FUNCTION_BLOCK FB_ProductHandling
VAR CONSTANT
	sCycleStateTextDef: ARRAY[0..30]  OF STRING :=	
		['State 0: Wait for Start',
		'State 1: Gantry A, Gantry B and Product conveyor started',
		'State 2: ',
		'3',
		'4',
		'5',
		'6',
		'7',
		'8',
		'9',
		'State 10:',
		'State 11:',
		'State 12:',
		'State 13:',
		'State 14:',
		'State 15:',
		'State 16:',
		'State 17:',
		'State 18:',
		'State 19:',
		'State 20: Stopcylce waiting for EAMC ready',
		'State 21: Stop cycle awaiting gantries ready',
		'State 22: Stop cycle awaiting outfeed conveyor ready',
		'State 23: Stop cycle Stopping Gantries and conveyor',
		'State 24: Stop cycle awaiting restart',
		'State 25: Stop direct'];
	
	tCycleStateTimeouts: ARRAY[0..10] OF TIME := 
		[T#10S,T#10S,T#10S,T#10S,T#10S,T#10S,T#10S,T#10S,T#10S,T#10S,
		T#10S];

	sInitStateTextDef: ARRAY[0..10] OF STRING :=
		['State 0: Wait for Start',
		'State 1: Description Init State 1',
		'State 2: Description Init State 2',
		'State 3; Description Init State 3',
		'State 4; Description Init State 4',
		'State 5; Description Init State 5',
		'State 6; Error State'];

	tInitStateTimeouts: ARRAY[0..10] OF TIME := 
		[T#10S,T#10S,T#10S,T#10S,T#10S,T#10S,T#10S,T#10S,T#10S,T#10S
		,T#10S];
END_VAR
VAR_INPUT
	mxResetCycleState				: BOOL;
	mxResetInitState				: BOOL;
	mxForceInit						: BOOL; (*Reset Calibration Flag*)
	mxReset							: BOOL;	(*Reset Error*)
	mxEmergency						: ARRAY [1..Max_Zones+1] OF BOOL; // 1=TakeOutA, 2=Aside, 3=mid, 4=Bside, 5=TakeoutB, 6= GantryB, 7=GantryA, 8=All EM stop.
	mxAutoMode						: BOOL; (* TRUE = Automode *)
	mxFirstCycle					: BOOL;
	mxSideA_Enabled					: BOOL;
	mxSideB_Enabled					: BOOL;
	mxEamcIsEmpty					: BOOL;
	mxProductReadyAtTakeout_A		: BOOL;
	mxProductReadyAtTakeout_B		: BOOL;
	
	mxPause							: BOOL;
END_VAR
VAR_IN_OUT
	MachParameters					: ST_ProductHandlingMachPar;
	ProdParameters					: ST_ProductHandlingProdPar;
	SysParameters					: ST_ProductHandlingSysPar;
END_VAR
VAR_OUTPUT
(*Errors*)
	Errors							: ST_ProductHandlingErrors;
	mxErrorInit						: BOOL;		(* Error, stop immediately. Initialisation neccesary *)
	mxErrorStopinPos				: BOOL;		(* Error, stop in position. Only reset neccesary *)

(* State vars *)
	mxCycleBusy						: BOOL;
	mxInitBusy						: BOOL;
	
(* Vars *)
	mxInitialized					: BOOL;
	mxProductPickedUpGantry_A		: BOOL;
	mxProductPickedUpGantry_B		: BOOL;
	mxGantrysNotBusy				: BOOL;
	
END_VAR
VAR
	(* State vars *)
	miCycleState					: INT :=0;
	miCycleOldstate					: INT :=0;
	mxCycleTransitionState			: BOOL := FALSE;
	sCycleStateText					: STRING;
	exCycleTimeOut					: BOOL;		(* Timeout for the whole programcycle *)
	CycleTimeout					: TON;
	CycleTimeOutUpFlank				: R_TRIG;
	mxCycleTimeoutEnable			: BOOL;
	CycleTime						: REAL;
	mxCycleHasError					: BOOL;
	miStopState						: INT;
	mxStartCycle					: BOOL;
	mxStopCycle						: BOOL;
	mxStopDirect					: BOOL;
	
	miInitState						: INT	:=0;
	miInitOldstate					: INT	:=0;
	mxInitTransitionState			: BOOL	:= FALSE;
	sInitStateText					: STRING;
	exInitTimeOut					: BOOL;		(* Timeout for the whole programcycle *)
	InitTimeout						: TON;
	InitTimeOutUpFlank				: R_TRIG;
	mxInitTimeoutEnable				: BOOL;
	InitTime						: REAL;
	mxInitHasError					: BOOL;
	mxStartInit						: BOOL;
	mxStopInit						: BOOL;

	(*Errors *)
	SR_HorMovingVertNotAtTranspPos_A	: SR;(* RedHot SafetyRule, Horizontal is moving when vertical is not at transport position *)
	SR_HorMovingVertNotAtTranspPos_B	: SR;(* RedHot SafetyRule, Horizontal is moving when vertical is not at transport position *)
	SR_VertMovingHorNotInPos_A			: SR;(* RedHot SafetyRule, Vertical is moving when horizontal is not at pick or drop position *)
	SR_VertMovingHorNotInPos_B			: SR;(* RedHot SafetyRule, Vertical is moving when horizontal is not at pick or drop position *)

	(* Objects *)
	GantryA								: FB_Gantry;
	GantryB								: FB_Gantry;
	OutfeedConveyor						: FB_OutfeedConveyor;
	
	mxHMI_DisableCollision				: BOOL;

	RT_ProductReadyAtTakeout_A: R_TRIG;
	RT_ProductReadyAtTakeout_B: R_TRIG;
	mxHorOnPos_A: BOOL;
	mxHorOnPos_B: BOOL;
	
	RT_AutoMode: R_TRIG;
	mxSafetyRulesEnabled: BOOL;
	T_StopCommisioningMode: TON;
	mxVertOnPos_A: BOOL;
	mxVertOnPos_B: BOOL;
	mxStopCycleEmpty: BOOL;
	
	
	mxInPause : BOOL;
END_VAR

(* Stopcycle = empty machine *)
(* Pause = stop at place *)

Error();
Cycle();
Init();
Objects();

RT_AutoMode(CLK:= mxAutoMode);
IF RT_AutoMode.Q THEN
	mxHMI_DisableCollision:= FALSE;
END_IF

T_StopCommisioningMode(IN:=MachParameters.CommisioningMode, PT:=T#120M);
IF T_StopCommisioningMode.Q THEN
	MachParameters.CommisioningMode := FALSE;
END_IF

ACTION Cycle:
(*StateChange (Transition)  Signalgeneration*)
mxCycleTransitionState:=(miCycleState<>miCycleOldstate);
(*State text*)
sCycleStateText:=sCycleStateTextDef[miCycleState];
(*Timeout Watchdog for Statemachine*)
mxCycleTimeoutEnable:=NOT (miCycleState=0) AND NOT mxReset;

CycleTimeout(IN:=mxCycleTimeoutEnable, PT:=tCycleStateTimeouts[miCycleState] );
CycleTimeOutUpFlank(CLK:=CycleTimeout.Q );
miCycleOldstate:=miCycleState;

(*Set Errorbit when Raising edge of Timeout has been detected*)
IF CycleTimeOutUpFlank.Q THEN
	exCycleTimeOut:=TRUE; 			(* 1 Timeout for the whole programcycle *)
END_IF

(*Function to reset the Statemachine*)
IF mxResetCycleState THEN
	mxResetCycleState:= FALSE;
	miCycleState:=0;
	miCycleOldstate:=miCycleState;
	mxCycleTransitionState:=FALSE;

	mxInitialized:= FALSE;
	mxStartCycle:= FALSE;
	mxStopCycle:= FALSE;
	mxStopCycleEmpty := FALSE;
	mxStopDirect:= FALSE;

	mxEamcIsEmpty:= FALSE;
	mxPause:= FALSE;
			
	GantryA.mxResetCycleState:= TRUE;
	GantryB.mxResetCycleState:= TRUE;
	OutfeedConveyor.mxResetCycleState:= TRUE;

END_IF

(*Definition State has Error*)
mxCycleHasError:=FALSE;

RT_ProductReadyAtTakeout_A(CLK:= mxProductReadyAtTakeout_A);
RT_ProductReadyAtTakeout_B(CLK:= mxProductReadyAtTakeout_B);

(*Cycle State's*)
CASE miCycleState OF
	0:
	(*
		- Wait for startcycle
		- Start GantryA, B, Outfeedconveyor

	Als Stop dan leegdraaien, dus wachten op EAMC die leeg is
	Als Pause dan alles stopInPos en vrijgeven. 
		*  
	*)
		IF mxStartCycle THEN
			mxStartCycle:= FALSE;

			IF mxSideA_Enabled THEN GantryA.M_StartCycle(); END_IF
			IF mxSideB_Enabled THEN GantryB.M_StartCycle(); END_IF
			OutfeedConveyor.M_StartCycle();
			
			miCycleState:= 1;
		END_IF	

	(* Gantry A, Gantry B, Outfeed started *)
	1:
		IF RT_ProductReadyAtTakeout_A.Q THEN
			GantryA.mxProductReadyAtTakeout:= TRUE;
		END_IF
		IF RT_ProductReadyAtTakeout_B.Q THEN
			GantryB.mxProductReadyAtTakeout:= TRUE;
		END_IF
	
		IF mxStopCycleEmpty AND mxEamcIsEmpty THEN (* Emtpy *)
			mxStopCycleEmpty:= FALSE;
			
			miStopState:= miCycleState;
			miCycleState:= 20;
		ELSIF mxStopCycle THEN
			mxStopCycle:= FALSE;			

			(* Stop Cycle *)
			IF mxSideA_Enabled THEN GantryA.M_StopCycle(); END_IF
			IF mxSideB_Enabled THEN GantryB.M_StopCycle(); END_IF
			OutfeedConveyor.M_StopCycle();
			
			miStopState:= miCycleState;
			miCycleState:= 23;
		END_IF

	(* Stop Cycle, wait for EAMC is empty *)
	20:
		IF mxStopDirect THEN
			mxStopDirect:= FALSE;
			
			miCycleState:= 25;
		ELSIF mxEamcIsEmpty THEN // Signal from EAMC that the machine is empty, Gantry A B signals are set when product ready at gantry
		
			miCycleState:= 21;			
		END_IF

	(* Stop Cycle, wait for Gantry is empty *)
	21:
		IF mxStopDirect THEN
			mxStopDirect:= FALSE;
			
			miCycleState:= 25;
		ELSIF (GantryA.mxIsEmpty OR NOT mxSideA_Enabled) AND (GantryB.mxIsEmpty OR NOT mxSideB_Enabled) THEN
		
			(* Stop Cycle *)
			IF mxSideA_Enabled THEN GantryA.M_StopCycle(); END_IF
			IF mxSideB_Enabled THEN GantryB.M_StopCycle(); END_IF
			OutfeedConveyor.M_StopCycle();
			
			miCycleState:= 22;
		END_IF

	(* Stop Cycle, outfeed conveyor empty *)
	22:
		IF mxStopDirect THEN
			mxStopDirect:= FALSE;
			
			miCycleState:= 25;
		ELSIF NOT OutfeedConveyor.mxCycleBusy THEN
		
			miCycleState:= 0;
		END_IF
	
	(* Stop Cycle, Stop gantry's, Belt *)
	23:
		IF mxStopDirect THEN
			mxStopDirect:= FALSE;
			
			miCycleState:= 25;
		ELSIF NOT GantryA.mxCycleBusy AND NOT GantryB.mxCycleBusy AND NOT OutfeedConveyor.mxCycleBusy THEN
			
			miCycleState:= 24;
		END_IF

	(* Stop Cycle, wait for restart *)
	24:
		IF mxStopDirect THEN
			mxStopDirect:= FALSE;
			
			miCycleState:= 25;
		ELSIF mxStartCycle THEN
			mxStartCycle:= FALSE;
			
			miCycleState:= miStopState;
		END_IF

	(* Stop Direct *)
	25:
		mxInitialized:= FALSE;
		mxStartCycle:= FALSE;
		mxStopCycle:= FALSE;
		mxStopDirect:= FALSE;

		GantryA.M_StopDirect();
		GantryB.M_StopDirect();
		OutfeedConveyor.M_StopDirect();
		
		miCycleState:= 0;
END_CASE

mxCycleBusy:= miCycleState<>0 AND NOT (miCycleState=22);
END_ACTION

ACTION Error:
(* Red Hot Safety *)

mxSafetyRulesEnabled := (mxInitialized AND mxAutoMode) OR (NOT mxAutomode); //AND NOT MachParameters.CommisioningMode;

mxHorOnPos_A:= (GantryA.mrActPosHorizontal <= (MachParameters.GantryA.PositionHorizontalPickup + 10) AND GantryA.mrActPosHorizontal >= (MachParameters.GantryA.PositionHorizontalPickup - 10)) OR
	 	(GantryA.mrActPosHorizontal <= (MachParameters.GantryA.PositionHorizontalDropOff + 10) AND GantryA.mrActPosHorizontal >= (MachParameters.GantryA.PositionHorizontalDropOff - 10));

mxHorOnPos_B:=(GantryB.mrActPosHorizontal <= (MachParameters.GantryB.PositionHorizontalPickup + 10) AND GantryB.mrActPosHorizontal >= (MachParameters.GantryB.PositionHorizontalPickup - 10)) OR
	 	(GantryB.mrActPosHorizontal <= (MachParameters.GantryB.PositionHorizontalDropOff + 10) AND GantryB.mrActPosHorizontal >= (MachParameters.GantryB.PositionHorizontalDropOff - 10));

mxVertOnPos_A := (GantryA.mrActPosVertical <= (MachParameters.GantryA.Vert_PositionTransport - 10) AND GantryA.mrActPosVertical >= (MachParameters.GantryA.Vert_PositionTransport + 5));

mxVertOnPos_B := (GantryB.mrActPosVertical <= (MachParameters.GantryB.Vert_PositionTransport - 10) AND GantryB.mrActPosVertical >= (MachParameters.GantryB.Vert_PositionTransport + 5));
		


SR_HorMovingVertNotAtTranspPos_A(
	SET1:= mxSafetyRulesEnabled AND mxAutoMode AND GantryA.mxHorizontalIsMoving AND mxVertOnPos_A, 
	RESET:= mxReset, Q1=> Errors.RH_HorMovingVertNotAtTranspPos_A);
	
SR_HorMovingVertNotAtTranspPos_B(
	SET1:=mxSafetyRulesEnabled AND mxAutoMode AND GantryB.mxHorizontalIsMoving AND mxVertOnPos_B,
	RESET:= mxReset, Q1=> Errors.RH_HorMovingVertNotAtTranspPos_B);

SR_VertMovingHorNotInPos_A(
	SET1:=mxSafetyRulesEnabled AND mxAutoMode AND GantryA.mxVerticalIsMoving AND NOT mxHorOnPos_A, 
	RESET:= mxReset, Q1=> Errors.RH_VertMovingHorNotInPos_A);

SR_VertMovingHorNotInPos_B(
	SET1:=mxSafetyRulesEnabled AND mxAutoMode AND GantryB.mxVerticalIsMoving AND NOT mxHorOnPos_B, 
	RESET:= mxReset, Q1=> Errors.RH_VertMovingHorNotInPos_B);

(*************************************************************************************************)
mxErrorInit:= GantryA.mxErrorInit OR GantryB.mxErrorInit OR OutfeedConveyor.mxErrorInit OR 
				Errors.RH_HorMovingVertNotAtTranspPos_A OR Errors.RH_HorMovingVertNotAtTranspPos_B OR 
				Errors.RH_VertMovingHorNotInPos_A OR Errors.RH_VertMovingHorNotInPos_B;
				
mxErrorStopinPos:= GantryA.mxErrorStopinPos OR GantryB.mxErrorStopinPos OR OutfeedConveyor.mxErrorStopinPos;
END_ACTION

ACTION Init:
(*StateChange (Transition)  Signalgeneration*)
mxInitTransitionState:=(miInitState<>miInitOldstate);
(*State text*)
sInitStateText:=sInitStateTextDef[miInitState];
(*Timeout Watchdog for Statemachine*)
mxInitTimeoutEnable:=NOT (miInitState=0)  AND NOT mxReset;

InitTimeout(IN:=mxInitTimeoutEnable  , PT:=tInitStateTimeouts[miInitState] );
InitTimeOutUpFlank(CLK:=InitTimeout.Q );
miInitOldstate:=miInitState;

(*Set Errorbit when Raising edge of Timeout has been detected*)
IF InitTimeOutUpFlank.Q THEN
	exInitTimeOut:=TRUE; 			(* 1 Timeout for the whole programcycle *)
END_IF

(*Function to reset the Statemachine*)
IF mxResetInitState THEN
	mxResetInitState:=FALSE;
	miInitState:=0;
	miInitOldstate:=miInitState;
	mxInitTransitionState:=FALSE;

	mxInitialized:= FALSE;
	mxStartInit:= FALSE;
	mxStopInit:= FALSE;
	
	GantryA.mxResetInitState:= TRUE;
	GantryA.mxResetCycleState:=TRUE;
	GantryB.mxResetInitState:=TRUE;
	GantryB.mxResetCycleState:= TRUE;
	OutFeedConveyor.mxResetInitState:=TRUE;
	OutfeedConveyor.mxResetCycleState:= TRUE;	
END_IF

(*Definition State has Error*)
mxInitHasError:=FALSE;

(*Init State's*)
CASE miInitState OF
	0:
	
	(* 
		- Wait for start int
		- Blow off uit
		- vacuum aan laten
		- Vertical move up to transport pos.
		- Horizontal move back to drop off positie
		- 	
	
	*)
		IF mxStartInit THEN
			mxStartInit:= FALSE;
			mxInitialized:= FALSE;
		
			miInitState:= 1;
		END_IF

	1:
		IF mxStopInit THEN
			mxStopInit:= FALSE;
			miInitState:= 10;
		ELSE
			IF mxSideA_Enabled THEN GantryA.M_StartInit(); END_IF			
			IF mxSideB_Enabled THEN GantryB.M_StartInit(); END_IF
			OutfeedConveyor.M_StartInit();

			miInitState:= 2;
		END_IF

	2:
		IF mxStopInit THEN
			mxStopInit:= FALSE;
			miInitState:= 10;
		ELSIF (GantryA.mxInitialized OR NOT mxSideA_Enabled) AND (GantryB.mxInitialized OR NOT mxSideB_Enabled)
				 AND OutfeedConveyor.mxInitialized THEN
	
			mxInitialized:= TRUE;
			miInitState:= 0;
		END_IF

	(* Stop Init *)
	10:
		mxStartInit:= FALSE;
		mxStopInit:= FALSE;
		mxInitialized:= FALSE;

		GantryA.M_StopInit();
		GantryB.M_StopInit();
		OutfeedConveyor.M_StopInit();
		
		miInitState:= 0;
			
END_CASE

mxInitBusy:= miInitState<>0;
END_ACTION

METHOD M_StartCycle

IF (NOT mxCycleBusy AND mxInitialized) OR (mxInPause AND mxInitialized) THEN
	mxInPause:=FALSE;
	mxStartCycle:= TRUE;	
END_IF
END_METHOD

METHOD M_StartInit

IF NOT mxInitBusy THEN 
	mxStartInit:= TRUE; 
END_IF
END_METHOD

METHOD M_StopCycle

IF mxCycleBusy THEN
	mxStopCycle:= TRUE;	
	mxInPause:=TRUE;
END_IF
END_METHOD

METHOD M_StopCycleEmpty

IF mxCycleBusy THEN 
	mxStopCycleEmpty:= TRUE; 
END_IF
END_METHOD

METHOD M_StopDirect

IF mxCycleBusy THEN
	mxStopDirect:= TRUE;	
END_IF
END_METHOD

METHOD M_StopInit

IF mxInitBusy THEN 
	mxStopInit:= TRUE; 
END_IF
END_METHOD

ACTION Objects:
GantryA(
	mxReset:= mxReset, 
	mxEmergency:= mxEmergency[1] OR mxEmergency[2] OR mxEmergency[7], 
	mxAutoMode:= mxAutoMode, 
	mxFirstCycle:= mxFirstCycle,
	mrModPosConveyor:= OutfeedConveyor.mrActModPos, 
	mxDisableCollision:= mxHMI_DisableCollision,
	MachParameters:= MachParameters.GantryA, 
	ProdParameters:= ProdParameters.GantryA, 
	SysParameters:= SysParameters.GantryA,
	mxProductPickedUp=> mxProductPickedUpGantry_A,
	Errors=> Errors.Gantry_A);
	
GantryB(
	mxReset:= mxReset, 
	mxEmergency:= mxEmergency[4] OR mxEmergency[5] OR mxEmergency[6], 
	mxAutoMode:= mxAutoMode, 
	mxFirstCycle:= mxFirstCycle,
	mrModPosConveyor:= OutfeedConveyor.mrActModPos, 
	mxDisableCollision:= mxHMI_DisableCollision,
	MachParameters:= MachParameters.GantryB, 
	ProdParameters:= ProdParameters.GantryB, 
	SysParameters:= SysParameters.GantryB,
	mxProductPickedUp=> mxProductPickedUpGantry_B,
	Errors=> Errors.Gantry_B);
	
OutfeedConveyor(
	mxReset:= mxReset, 
	mxEmergency:= mxEmergency[6] OR mxEmergency[7], 
	mxAutoMode:= mxAutoMode, 
	mxFirstCycle:= mxFirstCycle,
	MachParameters:= MachParameters.OutfeedConveyor, 
	ProdParameters:= ProdParameters.OutfeedConveyor, 
	SysParameters:= SysParameters.OutfeedConveyor,
	Errors=> Errors.OutfeedConveyor);
	
mxGantrysNotBusy:= NOT GantryA.mxCycleBusy AND NOT GantryB.mxCycleBusy;
END_ACTION

END_FUNCTION_BLOCK

(* stored: Version 1.1.0.1, ProductVersion 3.1.4020.12
   POU FB_ProductHandling: Id {61de353f-0cec-4382-8e02-a7518d515835}, SpecialFunc None
   Action Cycle: Id {5be5b63a-ceb4-4b96-8e47-4b368e0f91ea}
   Action Error: Id {e615a34a-f660-42d0-9760-54b009b1a521}
   Action Init: Id {28d39330-ecd3-4938-9695-4302f44b711e}
   Method M_StartCycle: Id {9dbb3887-6403-4c5f-a702-07955d178a78}
   Method M_StartInit: Id {8a591344-d71f-4a1f-8b2b-f21894e7e0b5}
   Method M_StopCycle: Id {0463aae5-2c23-4a89-adb3-cdf69b70a106}
   Method M_StopCycleEmpty: Id {2b14915f-953a-44d2-99d9-b6fbd415fed7}
   Method M_StopDirect: Id {a5105357-9460-4ce2-a9d5-da894fcb2c6f}
   Method M_StopInit: Id {8661507e-1601-449f-b1ad-4a175641e7b4}
   Action Objects: Id {25755bf5-e8da-4a8a-9179-61afed6531fc} *)
